PROGRAM MAIN
VAR
	m0 : DriverSequence();
	m1 : DriverSequence();
	
	enable : BOOL := TRUE;
	
	ready : BOOL;
	contUp : BOOL;
	contDown : BOOL;
	target : REAL := -1;
	
	auto : BOOL := TRUE;
	
	step : INT;
	timer : TON;
END_VAR

IF m0.ready AND m1.ready AND auto THEN
	autoSequence();
END_IF

m0(
	enable:= enable,
	contUp:= contUp, 
	contDown:= contDown, 
	target:= target,
	ready=> );

m1(
	enable:= enable,
	contUp:= contUp, 
	contDown:= contDown, 
	target:= target,
	ready=> );
	
(*
this module contains 2 ClearLink MC Motors
motors can be controlled manually or with an automatic demo routine
motors must be enabled and homed before use

contUp - continuous positive direction
contDown - continuous negative direction

target - target a specified position >= 0
*)

METHOD autoSequence : BOOL
VAR_INPUT
END_VAR
timer(IN:= , PT:= , Q=> , ET=> );

CASE step OF
	0: //+continuous for 5s
		timer.IN := TRUE;
		timer.PT := T#5S;
		
		contUp := TRUE;
		
		IF timer.Q THEN
			timer.IN := FALSE;
			contUp := FALSE;
			step := 10;
		END_IF
		
	10: //target
		IF m0.position = 150 AND NOT m0.busy AND m1.position = 150 AND NOT m1.busy THEN
			target := -1;
			step := 20;
			RETURN;
		END_IF
		
		target := 150;
		
		IF m0.busy AND m1.busy THEN
			//step := 11;
		END_IF
		
	11:
		//
	
	20: //-continuous 2s
		timer.IN := TRUE;
		timer.PT := T#2S;
		
		contDown := TRUE;
		
		IF timer.Q THEN
			timer.IN := FALSE;
			contDown := FALSE;
			step := 30;
		END_IF
	
	
	30: //target 0
		target := 0;
		
		IF m0.busy AND m1.busy THEN
			step := 31;
		END_IF
		
	31:
		IF m0.position = 0 AND NOT m0.busy AND m1.position = 0 AND NOT m1.busy THEN
			target := -1;
			step := 40;
			RETURN;
		END_IF
		
	40:
		timer.IN := TRUE;
		timer.PT := T#1S;
		
		IF timer.Q THEN
			timer.IN := FALSE;
			step := 0;
		END_IF
END_CASE
END_METHOD

END_PROGRAM

(* stored: Version 1.1.0.1, ProductVersion 3.1.4024.11
   POU MAIN: Id {13d21215-9747-4cee-a40e-9344284ff151}, SpecialFunc None
   Method autoSequence: Id {4f1817ea-dc64-469d-b2fa-6c14eaa3d76c} *)
